// TIA Portal project "Ex4-ControlCircuits" (V15.1)

(* hardware
DEVICE "S7-1200 station_1"  S7-1200 Station
   slot 0: "Rack_0"  S7-1200 Rack  Rack  V1.0
   slot 1: "PLC_1"  CPU 1215C DC/DC/Rly  6ES7 215-1HG40-0XB0  V4.2
*)

// ===== PLC "PLC_1"  CPU 1215C DC/DC/Rly =====

VAR_GLOBAL   // PLC tag table "Default tag table"
   "System_Byte" AT %MB254 : Byte;
   "FirstScan" AT %M254.0 : Bool;
   "DiagStatusUpdate" AT %M254.1 : Bool;
   "AlwaysTRUE" AT %M254.2 : Bool;
   "AlwaysFALSE" AT %M254.3 : Bool;
   "System_Byte(1)" AT %MB1 : Byte;
   "Clock_Byte" AT %MB255 : Byte;
   "Clock_10Hz" AT %M255.0 : Bool;
   "Clock_5Hz" AT %M255.1 : Bool;
   "Clock_2.5Hz" AT %M255.2 : Bool;
   "Clock_2Hz" AT %M255.3 : Bool;
   "Clock_1.25Hz" AT %M255.4 : Bool;
   "Clock_1Hz" AT %M255.5 : Bool;
   "Clock_0.625Hz" AT %M255.6 : Bool;
   "Clock_0.5Hz" AT %M255.7 : Bool;
   "iCC_BtnStop_S1" AT %I0.0 : Bool;   // Red stop push button
   "iCC_BtnStart_S3" AT %I0.2 : Bool;   // Green start push button
   "mStarted_H1" AT %M0.0 : Bool;   // Installation 1 started
   "mStarted_H2" AT %M0.1 : Bool;   // Installation 2 started
   "oCC_LmpStart_H1" AT %Q0.0 : Bool;   // Green lamp installation 1 started
   "oCC_LmpStart_H2" AT %Q0.1 : Bool;   // Green lamp installation 2 started
   "iCC_BtnReset_S5" AT %I0.4 : Bool;   // Reset pushbutton
   "iCC_MbcMot_QM1" AT %I0.6 : Bool;   // Motor circuit breaker feedback signal
   "mA001" AT %M2.0 : Bool;   // Circuit breaker failure motor 1 [-M1]
   "mA001_016" AT %MW2 : Word;   // Alarms 001 to 016
   "oCC_ConMot_KM1" AT %Q0.6 : Bool;   // Motor contactor [-M1]
   "oCC_LmpTest_H3" AT %Q0.2 : Bool;   // Yellow lamp - Teleruptor test
   "iCC_BtnTest_S4" AT %I0.3 : Bool;   // Teleruptor test push button
   "mCC_PoBtnTest_S4" AT %M0.2 : Bool;   // Rising edge on iCC1_BtnTest_S4
   "mTelrup_H3" AT %M0.3 : Bool;   // Teleruptor H3
END_VAR

FUNCTION "FC_StartStop" : Void   // FC1, FBD
TITLE = Start stop circuits
{ S7_Optimized_Access := 'TRUE' }
VERSION : 0.1
BEGIN

REGION Network 1: Start-stop circuit (FlipFlop)
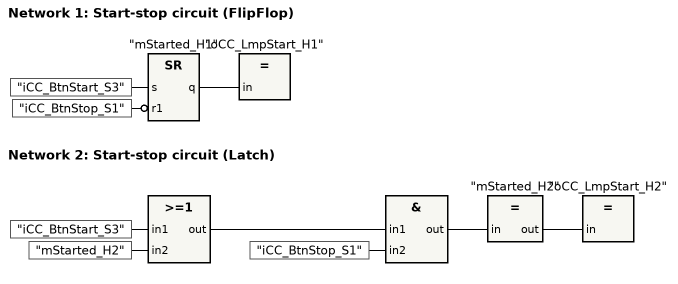
   IF "iCC_BtnStart_S3" THEN
       "mStarted_H1" := TRUE;   // SR flip-flop
   END_IF;
   IF NOT "iCC_BtnStop_S1" THEN "mStarted_H1" := FALSE; END_IF;
   "oCC_LmpStart_H1" := "mStarted_H1";
END_REGION

REGION Network 2: Start-stop circuit (Latch)
   "mStarted_H2" := ("iCC_BtnStart_S3" OR "mStarted_H2") AND "iCC_BtnStop_S1";
   "oCC_LmpStart_H2" := "mStarted_H2";
END_REGION
END_FUNCTION

FUNCTION "FC_Alarm" : Void   // FC2, FBD
TITLE = Alarm control circuit
{ S7_Optimized_Access := 'TRUE' }
VERSION : 0.1
BEGIN

REGION Network 1: Motor circuit breaker failure
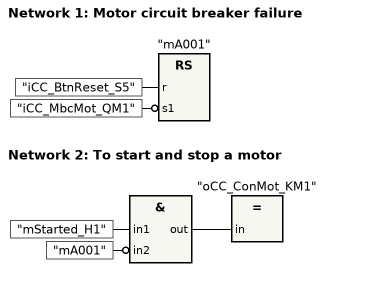
   IF "iCC_BtnReset_S5" THEN
       "mA001" := FALSE;   // RS flip-flop
   END_IF;
   IF NOT "iCC_MbcMot_QM1" THEN "mA001" := TRUE; END_IF;
END_REGION

REGION Network 2: To start and stop a motor
   "oCC_ConMot_KM1" := "mStarted_H1" AND NOT "mA001";
END_REGION
END_FUNCTION

FUNCTION "FC_Teleruptor" : Void   // FC3, FBD
TITLE = Teleruptor circuit
{ S7_Optimized_Access := 'TRUE' }
VERSION : 0.1
   VAR_TEMP   // added for the SCL form of the ladder/FBD networks
      _w1 : Bool;
   END_VAR
BEGIN

REGION Network 1: Test light point H3
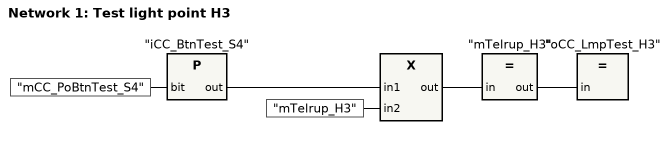
   #_w1 := "iCC_BtnTest_S4" AND NOT "mCC_PoBtnTest_S4";   // rising edge of "iCC_BtnTest_S4"
   "mCC_PoBtnTest_S4" := "iCC_BtnTest_S4";
   "mTelrup_H3" := #_w1 XOR "mTelrup_H3";
   "oCC_LmpTest_H3" := "mTelrup_H3";
END_REGION
END_FUNCTION

ORGANIZATION_BLOCK "Main"   // OB1, FBD, ProgramCycle
TITLE = "Main Program Sweep (Cycle)"
{ S7_Optimized_Access := 'TRUE' }
VERSION : 0.1
   VAR_INPUT
      Initial_Call : Bool;   // Initial call of this OB
      Remanence : Bool;   // =True, if remanent data are available
   END_VAR
BEGIN

REGION Network 1: Start stop circuits
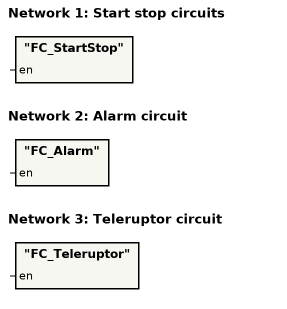
   "FC_StartStop"();
END_REGION

REGION Network 2: Alarm circuit
   "FC_Alarm"();
END_REGION

REGION Network 3: Teleruptor circuit
   "FC_Teleruptor"();
END_REGION
END_ORGANIZATION_BLOCK